(* Logix 5000 project; controller ThicknessMeasurement vendor 1 type 14 code 196 rev 33.11; software revision 33.00 *)

TASK MainTask (continuous, watchdog 500 ms) : MainProgram

MODULES
   Local : vendor 1 type 14 code 196 (5069 0, rev 33.11)
       : vendor 1 type 12 code 320 (5069 1, rev 2.12, StandardDataDriven RPI 80 ms, StandardDataDriven RPI 80 ms)
END_MODULES

VAR_GLOBAL   (* controller tags *)
   Comm_Error : COUNTER[13] := ([0].PRE := 3, [0].ACC := 1, [1].PRE := 3, [1].ACC := 1, [2].PRE := 3, [2].ACC := 1, [2].CU := 1, [3].PRE := 3, [3].ACC := 221, [3].DN := 1, [4].PRE := 3, [4].ACC := 226, [4].DN := 1, [5].PRE := 3, [5].ACC := 226, [5].DN := 1, [6].PRE := 3, [6].ACC := 218, [6].DN := 1, [7].PRE := 3, [7].ACC := 226, [7].DN := 1, [8].PRE := 3, [8].ACC := 226, [8].DN := 1, [9].PRE := 3, [9].ACC := 227, [9].DN := 1, [10].PRE := 3, [10].ACC := 227, [10].DN := 1, [11].PRE := 3, [11].ACC := 227, [11].DN := 1, [12].PRE := 3, [12].ACC := 227, [12].DN := 1);
   HMI_Thickness : REAL[13] := ([0] := -0.4028, [1] := -0.9222, [2] := -0.8096);
   Last_HMI_Thickness : REAL[13] := ([0] := -0.4028, [1] := -0.9222, [2] := -0.8096);
   Last_RxID : DINT := -83;
   Receive_String : STRING_32[13] := ([0] := '%01$$RMD-000402848$0D', [1] := '%02$$RMD-00092224E$0D', [2] := '%03$$RMD-000809643$0D', [3] := '%04$$RMD+146327949$0D', [4] := '%03$$RMD+01122804A$0D', [5] := '%03$$RMD+01122804A$0D', [6] := '%07$$RMD-00081074E$0D', [7] := '%03$$RMD+01122804A$0D', [8] := '%03$$RMD+01122804A$0D', [9] := '%03$$RMD+001811348$0D', [10] := '%03$$RMD+001811348$0D', [11] := '%03$$RMD+001811348$0D', [12] := '%03$$RMD+001811348$0D');
   Reference_Point : REAL[13] := ([0] := -0.4269, [1] := -0.9956, [2] := -0.8743);
   Sampling_Period : TIMER := (PRE := 1000, EN := 1, TT := 1);
   Send_String : STRING_32[13] := ([0] := '%01#RMD5C$0D', [1] := '%02#RMD5F$0D', [2] := '%03#RMD5E$0D', [3] := 'HMI_Thickness[0]', [4] := '%05#RMD58$0D', [5] := '%06#RMD5B$0D', [6] := '%07#RMD5A$0D', [7] := '%08#RMD55$0D', [8] := '%09#RMD54$0D', [9] := '%10#RMD5C$0D', [10] := '%11#RMD5D$0D', [11] := '%12#RMD5E$0D', [12] := '%13#RMD5F$0D');
   Set : BOOL;
   Set_Ref_Point : BOOL;
   Set_String : STRING_32[13] := ([0] := '%01#RMD5C$0D', [1] := '%02#RMD5F$0D', [2] := '%03#RMD5E$0D', [3] := '%04#RMD59$0D', [4] := '%05#RMD58$0D', [5] := '%06#RMD5B$0D', [6] := '%07#RMD5A$0D', [7] := '%08#RMD55$0D', [8] := '%09#RMD54$0D', [9] := '%10#RMD5C$0D', [10] := '%11#RMD5D$0D', [11] := '%12#RMD5E$0D', [12] := '%13#RMD5F$0D');
   Truncate_String : STRING_32[13] := ([0] := '-0004028', [1] := '-0009222', [2] := '-0008096', [3] := '+1463279', [4] := '+0112280', [5] := '+0112280', [6] := '-0008107', [7] := '+0112280', [8] := '+0112280', [9] := '+0112280', [10] := '+0018113', [11] := '+0018113', [12] := '+0018113');
   TS2DINT : DINT[13] := ([0] := -4028, [1] := -9222, [2] := -8096, [3] := 1463279, [4] := 112280, [5] := 112280, [6] := -8107, [7] := 112280, [8] := 112280, [9] := 112280, [10] := 18113, [11] := 18113, [12] := 18113);
   Update : BOOL[32] := ([2] := 1);
END_VAR

PROGRAM MainProgram   (* main routine MainRoutine *)

ROUTINE MainRoutine   (* ladder *)
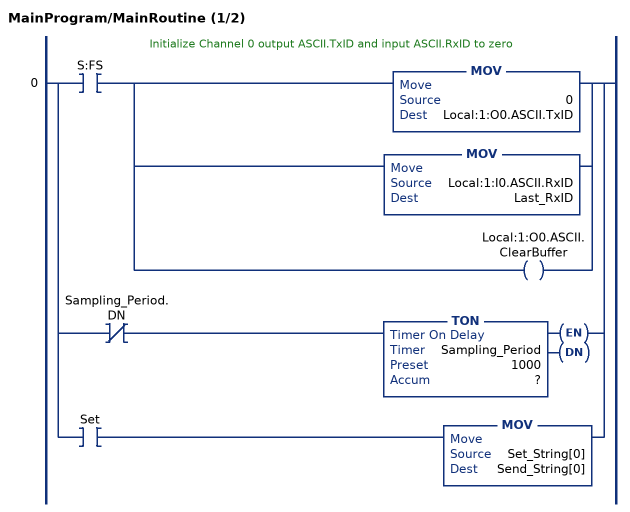
   // Initialize Channel 0 output ASCII.TxID and input ASCII.RxID to zero
   0: [XIC(S:FS) [MOV(0,Local:1:O0.ASCII.TxID) ,MOV(Local:1:I0.ASCII.RxID,Last_RxID) ,OTE(Local:1:O0.ASCII.ClearBuffer) ] ,XIO(Sampling_Period.DN) TON(Sampling_Period,?,?) ,XIC(Set) MOV(Set_String[0],Send_String[0]) ];
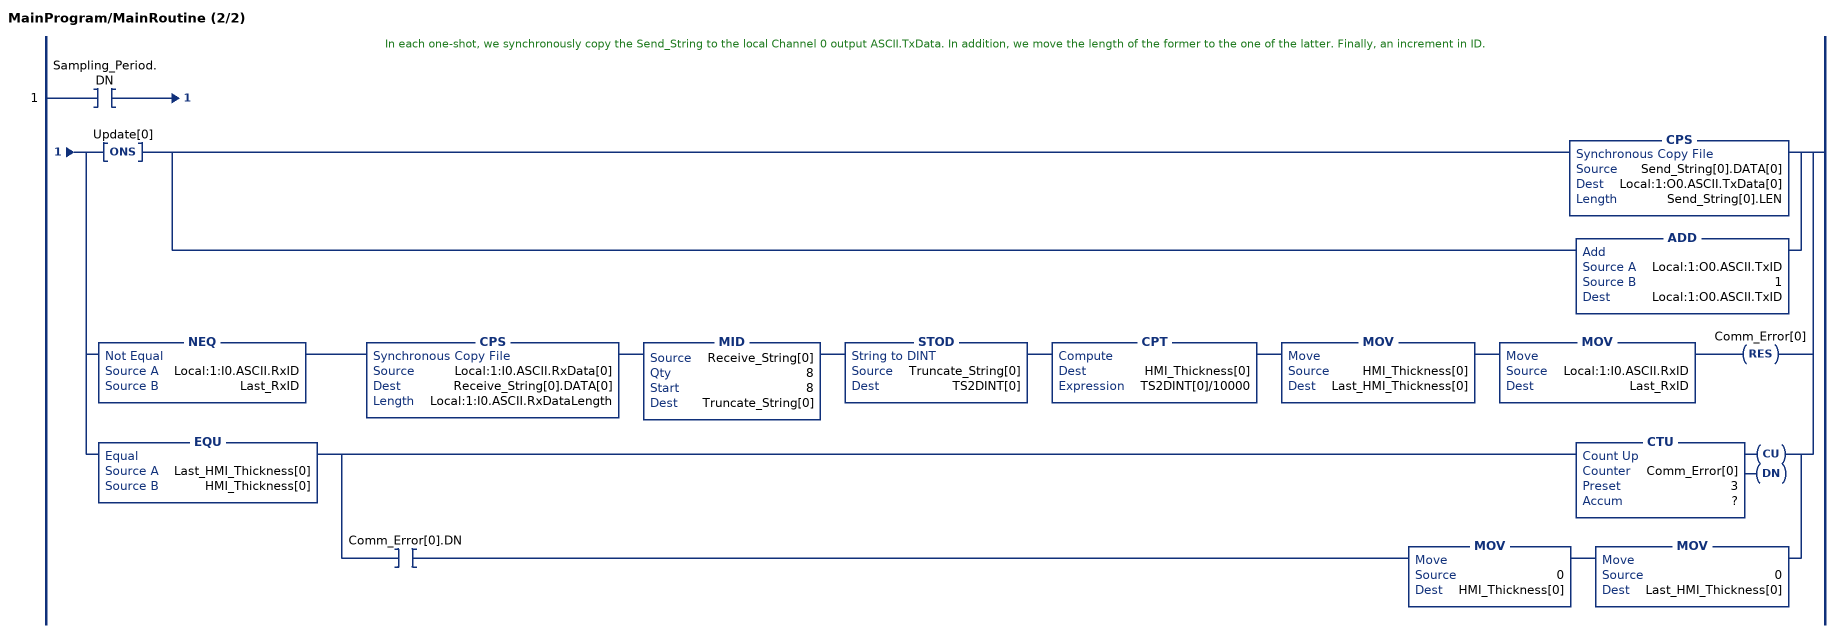
   // In each one-shot, we synchronously copy the Send_String to the local Channel 0 output ASCII.TxData. In addition, we move the length of the former to the one of the latter. Finally, an increment in ID.
   1: XIC(Sampling_Period.DN)[ONS(Update[0]) [CPS(Send_String[0].DATA[0],Local:1:O0.ASCII.TxData[0],Send_String[0].LEN) ,ADD(Local:1:O0.ASCII.TxID,1,Local:1:O0.ASCII.TxID) ] ,NEQ(Local:1:I0.ASCII.RxID,Last_RxID) CPS(Local:1:I0.ASCII.RxData[0],Receive_String[0].DATA[0],Local:1:I0.ASCII.RxDataLength) MID(Receive_String[0],8,8,Truncate_String[0]) STOD(Truncate_String[0],TS2DINT[0]) CPT(HMI_Thickness[0],TS2DINT[0]/10000) MOV(HMI_Thickness[0],Last_HMI_Thickness[0]) MOV(Local:1:I0.ASCII.RxID,Last_RxID) RES(Comm_Error[0]) ,EQU(Last_HMI_Thickness[0],HMI_Thickness[0]) [CTU(Comm_Error[0],?,?) ,XIC(Comm_Error[0].DN) MOV(0,HMI_Thickness[0]) MOV(0,Last_HMI_Thickness[0]) ] ];
END_ROUTINE
END_PROGRAM
